LIN {X 0,Y 77.962,Z 440.495,A -85,B 0,C 180,E1 -28389.126,E2 -28389.126} C_VEL
LIN {X 0,Y 84.259,Z 435.416,A -85,B 0,C 180,E1 -28395.152,E2 -28395.152} C_VEL
LIN {X 0,Y 91.354,Z 428.999,A -85,B 0,C 180,E1 -28400.293,E2 -28400.293} C_VEL
LIN {X 0,Y 98.775,Z 421.332,A -85,B 0,C 180,E1 -28404.517,E2 -28404.517} C_VEL
LIN {X 0,Y 99.783,Z 419.685,A -85,B 0,C 180,E1 -28405.704,E2 -28405.704} C_VEL
LIN {X 0,Y 94.04,Z 422.037,A -85,B 0,C 180,E1 -28408.457,E2 -28408.457} C_VEL
LIN {X 0,Y 84.561,Z 425.489,A -85,B 0,C 180,E1 -28415.445,E2 -28415.445} C_VEL
LIN {X 0,Y 74.4,Z 429.626,A -85,B 0,C 180,E1 -28429.11,E2 -28429.11} C_VEL
LIN {X 0,Y 70.741,Z 435.431,A -85,B 0,C 180,E1 -28457.34,E2 -28457.34} C_VEL
LIN {X 0,Y 72.341,Z 436.386,A -85,B 0,C 180,E1 -28462.867,E2 -28462.867} C_VEL
LIN {X 0,Y 74.062,Z 437.713,A -85,B 0,C 180,E1 -28468.324,E2 -28468.324} C_VEL
LIN {X 0,Y 85.261,Z 440.555,A -85,B 0,C 180,E1 -28482.705,E2 -28482.705} C_VEL
LIN {X 0,Y 85.617,Z 441.316,A -85,B 0,C 180,E1 -28484.089,E2 -28484.089} C_VEL
LIN {X 0,Y 79.44,Z 445.871,A -85,B 0,C 180,E1 -28488.431,E2 -28488.431} C_VEL
LIN {X 0,Y 73.09,Z 450.242,A -85,B 0,C 180,E1 -28494.765,E2 -28494.765} C_VEL
LIN {X 0,Y 69.721,Z 452.565,A -85,B 0,C 180,E1 -28499.734,E2 -28499.734} C_VEL
LIN {X 0,Y 67.029,Z 454.469,A -85,B 0,C 180,E1 -28505.203,E2 -28505.203} C_VEL
LIN {X 0,Y 65.013,Z 455.908,A -85,B 0,C 180,E1 -28511.077,E2 -28511.077} C_VEL
LIN {X 0,Y 63.097,Z 457.574,A -85,B 0,C 180,E1 -28523.605,E2 -28523.605} C_VEL
LIN {X 0,Y 63.171,Z 457.811,A -85,B 0,C 180,E1 -28530,E2 -28530} C_VEL
LIN {X 0,Y 62.977,Z 457.55,A -85,B 0,C 180,E1 -28536.407,E2 -28536.407} C_VEL
LIN {X 0,Y 64.541,Z 455.84,A -85,B 0,C 180,E1 -28549.067,E2 -28549.067} C_VEL
LIN {X 0,Y 66.371,Z 454.364,A -85,B 0,C 180,E1 -28555.06,E2 -28555.06} C_VEL
LIN {X 0,Y 70.506,Z 451.34,A -85,B 0,C 180,E1 -28563.247,E2 -28563.247} C_VEL
LIN {X 0,Y 76.044,Z 447.27,A -85,B 0,C 180,E1 -28570.312,E2 -28570.312} C_VEL
LIN {X 0,Y 84.031,Z 441.038,A -85,B 0,C 180,E1 -28577.039,E2 -28577.039} C_VEL
LIN {X 0,Y 86.611,Z 438.899,A -85,B 0,C 180,E1 -28578.715,E2 -28578.715} C_VEL
LIN {X 0,Y 87.079,Z 437.956,A -85,B 0,C 180,E1 -28579.784,E2 -28579.784} C_VEL
LIN {X 0,Y 79.619,Z 436.48,A -85,B 0,C 180,E1 -28588.02,E2 -28588.02} C_VEL
LIN {X 0,Y 77.169,Z 435.308,A -85,B 0,C 180,E1 -28592.912,E2 -28592.912} C_VEL
LIN {X 0,Y 73.406,Z 433.371,A -85,B 0,C 180,E1 -28603.308,E2 -28603.308} C_VEL
LIN {X 0,Y 73.693,Z 429.74,A -85,B 0,C 180,E1 -28620,E2 -28620} C_VEL
LIN {X 0,Y 88.317,Z 421.829,A -85,B 0,C 180,E1 -28643.446,E2 -28643.446} C_VEL
LIN {X 0,Y 103.173,Z 415.563,A -85,B 0,C 180,E1 -28653.021,E2 -28653.021} C_VEL
LIN {X 0,Y 101.741,Z 417.578,A -85,B 0,C 180,E1 -28654.011,E2 -28654.011} C_VEL
LIN {X 0,Y 93.912,Z 426.276,A -85,B 0,C 180,E1 -28658.207,E2 -28658.207} C_VEL
LIN {X 0,Y 89.203,Z 430.846,A -85,B 0,C 180,E1 -28661.199,E2 -28661.199} C_VEL
LIN {X 0,Y 85.408,Z 433.951,A -85,B 0,C 180,E1 -28663.392,E2 -28663.392} C_VEL
LIN {X 0,Y 77.909,Z 438.596,A -85,B 0,C 180,E1 -28666.616,E2 -28666.616} C_VEL
LIN {X 0,Y 70.452,Z 442.536,A -85,B 0,C 180,E1 -28670.669,E2 -28670.669} C_VEL
LIN {X 0,Y 66.915,Z 444.545,A -85,B 0,C 180,E1 -28674.23,E2 -28674.23} C_VEL
LIN {X 0,Y 61.91,Z 447.609,A -85,B 0,C 180,E1 -28682.994,E2 -28682.994} C_VEL
LIN {X 0,Y 59.524,Z 449.005,A -85,B 0,C 180,E1 -28689.255,E2 -28689.255} C_VEL
LIN {X 0,Y 57.76,Z 449.987,A -85,B 0,C 180,E1 -28695.916,E2 -28695.916} C_VEL
LIN {X 0,Y 56.313,Z 450.815,A -85,B 0,C 180,E1 -28710,E2 -28710} C_VEL
LIN {X 0,Y 56.662,Z 450.615,A -85,B 0,C 180,E1 -28717.125,E2 -28717.125} C_VEL
LIN {X 0,Y 57.758,Z 450.026,A -85,B 0,C 180,E1 -28724.085,E2 -28724.085} C_VEL
LIN {X 0,Y 59.479,Z 449.063,A -85,B 0,C 180,E1 -28730.762,E2 -28730.762} C_VEL
LIN {X 0,Y 61.849,Z 447.699,A -85,B 0,C 180,E1 -28737.035,E2 -28737.035} C_VEL
LIN {X 0,Y 66.64,Z 444.824,A -85,B 0,C 180,E1 -28745.454,E2 -28745.454} C_VEL
LIN {X 0,Y 72.59,Z 440.908,A -85,B 0,C 180,E1 -28752.666,E2 -28752.666} C_VEL
LIN {X 0,Y 79.422,Z 435.826,A -85,B 0,C 180,E1 -28758.778,E2 -28758.778} C_VEL
LIN {X 0,Y 86.994,Z 429.408,A -85,B 0,C 180,E1 -28763.889,E2 -28763.889} C_VEL
LIN {X 0,Y 88.776,Z 427.801,A -85,B 0,C 180,E1 -28764.882,E2 -28764.882} C_VEL
LIN {X 0,Y 89.809,Z 426.453,A -85,B 0,C 180,E1 -28766.067,E2 -28766.067} C_VEL
LIN {X 0,Y 77.142,Z 430.533,A -85,B 0,C 180,E1 -28775.651,E2 -28775.651} C_VEL
LIN {X 0,Y 66.265,Z 434.834,A -85,B 0,C 180,E1 -28793.912,E2 -28793.912} C_VEL
LIN {X 0,Y 68.672,Z 441.312,A -85,B 0,C 180,E1 -28830.778,E2 -28830.778} C_VEL
LIN {X 0,Y 75.605,Z 442.948,A -85,B 0,C 180,E1 -28840.594,E2 -28840.594} C_VEL
LIN {X 0,Y 76.773,Z 443.733,A -85,B 0,C 180,E1 -28842.917,E2 -28842.917} C_VEL
LIN {X 0,Y 69.583,Z 448.493,A -85,B 0,C 180,E1 -28848.965,E2 -28848.965} C_VEL
LIN {X 0,Y 63.675,Z 452.15,A -85,B 0,C 180,E1 -28856.505,E2 -28856.505} C_VEL
LIN {X 0,Y 60.649,Z 454.053,A -85,B 0,C 180,E1 -28862.386,E2 -28862.386} C_VEL
LIN {X 0,Y 58.345,Z 455.493,A -85,B 0,C 180,E1 -28868.816,E2 -28868.816} C_VEL
LIN {X 0,Y 56.039,Z 457.158,A -85,B 0,C 180,E1 -28882.795,E2 -28882.795} C_VEL
LIN {X 0,Y 56.073,Z 457.395,A -85,B 0,C 180,E1 -28890,E2 -28890} C_VEL
LIN {X 0,Y 55.912,Z 457.133,A -85,B 0,C 180,E1 -28897.221,E2 -28897.221} C_VEL
LIN {X 0,Y 57.849,Z 455.422,A -85,B 0,C 180,E1 -28911.375,E2 -28911.375} C_VEL
LIN {X 0,Y 59.973,Z 453.945,A -85,B 0,C 180,E1 -28917.953,E2 -28917.953} C_VEL
LIN {X 0,Y 64.68,Z 450.924,A -85,B 0,C 180,E1 -28926.7,E2 -28926.7} C_VEL
LIN {X 0,Y 70.763,Z 446.853,A -85,B 0,C 180,E1 -28934.045,E2 -28934.045} C_VEL
LIN {X 0,Y 77.918,Z 441.734,A -85,B 0,C 180,E1 -28939.843,E2 -28939.843} C_VEL
LIN {X 0,Y 78.192,Z 440.975,A -85,B 0,C 180,E1 -28941.011,E2 -28941.011} C_VEL
LIN {X 0,Y 74.5,Z 440.2,A -85,B 0,C 180,E1 -28945.527,E2 -28945.527} C_VEL
LIN {X 0,Y 66.846,Z 436.213,A -85,B 0,C 180,E1 -28967.862,E2 -28967.862} C_VEL
LIN {X 0,Y 67.704,Z 433.913,A -85,B 0,C 180,E1 -28980,E2 -28980} C_VEL
LIN {X 0,Y 79.471,Z 427.848,A -85,B 0,C 180,E1 -29001.484,E2 -29001.484} C_VEL
LIN {X 0,Y 88.577,Z 424.457,A -85,B 0,C 180,E1 -29009.216,E2 -29009.216} C_VEL
LIN {X 0,Y 93.109,Z 422.662,A -85,B 0,C 180,E1 -29011.896,E2 -29011.896} C_VEL
LIN {X 0,Y 92.428,Z 424.025,A -85,B 0,C 180,E1 -29013.237,E2 -29013.237} C_VEL
LIN {X 0,Y 84.454,Z 431.482,A -85,B 0,C 180,E1 -29017.761,E2 -29017.761} C_VEL
LIN {X 0,Y 77.146,Z 437.451,A -85,B 0,C 180,E1 -29023.214,E2 -29023.214} C_VEL
LIN {X 0,Y 70.515,Z 442.168,A -85,B 0,C 180,E1 -29029.621,E2 -29029.621} C_VEL
LIN {X 0,Y 66.915,Z 444.545,A -85,B 0,C 180,E1 -29034.23,E2 -29034.23} C_VEL
LIN {X 0,Y 63.619,Z 446.327,A -85,B 0,C 180,E1 -29038.239,E2 -29038.239} C_VEL
LIN {X 0,Y 57.223,Z 448.651,A -85,B 0,C 180,E1 -29045.088,E2 -29045.088} C_VEL
LIN {X 0,Y 52.565,Z 450.064,A -85,B 0,C 180,E1 -29051.716,E2 -29051.716} C_VEL
LIN {X 0,Y 50.038,Z 450.83,A -85,B 0,C 180,E1 -29058.873,E2 -29058.873} C_VEL
LIN {X 0,Y 49.868,Z 450.864,A -85,B 0,C 180,E1 -29059.987,E2 -29059.987} C_VEL
LIN {X 0,Y 49.322,Z 451.164,A -85,B 0,C 180,E1 -29074.082,E2 -29074.082} C_VEL
LIN {X 0,Y 50.919,Z 450.441,A -85,B 0,C 180,E1 -29086.025,E2 -29086.025} C_VEL
LIN {X 0,Y 52.911,Z 449.477,A -85,B 0,C 180,E1 -29093.483,E2 -29093.483} C_VEL
LIN {X 0,Y 55.633,Z 448.112,A -85,B 0,C 180,E1 -29100.352,E2 -29100.352} C_VEL
LIN {X 0,Y 61.005,Z 445.237,A -85,B 0,C 180,E1 -29109.318,E2 -29109.318} C_VEL
LIN {X 0,Y 67.54,Z 441.321,A -85,B 0,C 180,E1 -29116.752,E2 -29116.752} C_VEL
LIN {X 0,Y 74.945,Z 436.237,A -85,B 0,C 180,E1 -29122.853,E2 -29122.853} C_VEL
LIN {X 0,Y 78.943,Z 433.189,A -85,B 0,C 180,E1 -29125.47,E2 -29125.47} C_VEL
LIN {X 0,Y 79.597,Z 432.225,A -85,B 0,C 180,E1 -29126.908,E2 -29126.908} C_VEL
LIN {X 0,Y 68.902,Z 435.279,A -85,B 0,C 180,E1 -29136.635,E2 -29136.635} C_VEL
LIN {X 0,Y 57.879,Z 441.553,A -85,B 0,C 180,E1 -29174.055,E2 -29174.055} C_VEL
LIN {X 0,Y 63.243,Z 444.517,A -85,B 0,C 180,E1 -29193.754,E2 -29193.754} C_VEL
LIN {X 0,Y 67.631,Z 445.456,A -85,B 0,C 180,E1 -29200.255,E2 -29200.255} C_VEL
LIN {X 0,Y 66.833,Z 446.644,A -85,B 0,C 180,E1 -29202.599,E2 -29202.599} C_VEL
LIN {X 0,Y 59.883,Z 450.655,A -85,B 0,C 180,E1 -29209.797,E2 -29209.797} C_VEL
LIN {X 0,Y 54.436,Z 453.637,A -85,B 0,C 180,E1 -29218.908,E2 -29218.908} C_VEL
LIN {X 0,Y 51.768,Z 455.077,A -85,B 0,C 180,E1 -29225.966,E2 -29225.966} C_VEL
LIN {X 0,Y 49.953,Z 456.106,A -85,B 0,C 180,E1 -29233.657,E2 -29233.657} C_VEL
LIN {X 0,Y 48.992,Z 456.742,A -85,B 0,C 180,E1 -29241.752,E2 -29241.752} C_VEL
LIN {X 0,Y 48.958,Z 456.979,A -85,B 0,C 180,E1 -29250,E2 -29250} C_VEL
LIN {X 0,Y 48.85,Z 456.716,A -85,B 0,C 180,E1 -29258.272,E2 -29258.272} C_VEL
LIN {X 0,Y 51.266,Z 455.004,A -85,B 0,C 180,E1 -29274.284,E2 -29274.284} C_VEL
LIN {X 0,Y 53.767,Z 453.526,A -85,B 0,C 180,E1 -29281.524,E2 -29281.524} C_VEL
LIN {X 0,Y 59.139,Z 450.508,A -85,B 0,C 180,E1 -29290.815,E2 -29290.815} C_VEL
LIN {X 0,Y 65.834,Z 446.436,A -85,B 0,C 180,E1 -29298.355,E2 -29298.355} C_VEL
LIN {X 0,Y 67.932,Z 445.077,A -85,B 0,C 180,E1 -29300.149,E2 -29300.149} C_VEL
LIN {X 0,Y 69.391,Z 443.577,A -85,B 0,C 180,E1 -29302.578,E2 -29302.578} C_VEL
LIN {X 0,Y 60.743,Z 439.877,A -85,B 0,C 180,E1 -29326.621,E2 -29326.621} C_VEL
LIN {X 0,Y 61.47,Z 437.706,A -85,B 0,C 180,E1 -29340,E2 -29340} C_VEL
LIN {X 0,Y 77.657,Z 430.826,A -85,B 0,C 180,E1 -29366.905,E2 -29366.905} C_VEL
LIN {X 0,Y 82.569,Z 429.212,A -85,B 0,C 180,E1 -29370.711,E2 -29370.711} C_VEL
LIN {X 0,Y 83.06,Z 429.58,A -85,B 0,C 180,E1 -29372.205,E2 -29372.205} C_VEL
LIN {X 0,Y 75.013,Z 436.037,A -85,B 0,C 180,E1 -29377.215,E2 -29377.215} C_VEL
LIN {X 0,Y 67.597,Z 441.161,A -85,B 0,C 180,E1 -29383.299,E2 -29383.299} C_VEL
LIN {X 0,Y 61.052,Z 445.118,A -85,B 0,C 180,E1 -29390.718,E2 -29390.718} C_VEL
LIN {X 0,Y 55.681,Z 448.025,A -85,B 0,C 180,E1 -29399.677,E2 -29399.677} C_VEL
LIN {X 0,Y 52.966,Z 449.42,A -85,B 0,C 180,E1 -29406.542,E2 -29406.542} C_VEL
LIN {X 0,Y 49.868,Z 450.864,A -85,B 0,C 180,E1 -29419.987,E2 -29419.987} C_VEL
LIN {X 0,Y 48.641,Z 451.264,A -85,B 0,C 180,E1 -29426.696,E2 -29426.696} C_VEL
LIN {X 0,Y 46.119,Z 451.387,A -85,B 0,C 180,E1 -29438.326,E2 -29438.326} C_VEL
LIN {X 0,Y 45.232,Z 450.886,A -85,B 0,C 180,E1 -29448.299,E2 -29448.299} C_VEL
LIN {X 0,Y 46.124,Z 450.089,A -85,B 0,C 180,E1 -29455.631,E2 -29455.631} C_VEL
LIN {X 0,Y 46.809,Z 449.734,A -85,B 0,C 180,E1 -29457.89,E2 -29457.89} C_VEL
LIN {X 0,Y 49.659,Z 448.525,A -85,B 0,C 180,E1 -29464.479,E2 -29464.479} C_VEL
LIN {X 0,Y 55.699,Z 445.65,A -85,B 0,C 180,E1 -29473.946,E2 -29473.946} C_VEL
LIN {X 0,Y 62.893,Z 441.733,A -85,B 0,C 180,E1 -29481.464,E2 -29481.464} C_VEL
LIN {X 0,Y 68.149,Z 438.461,A -85,B 0,C 180,E1 -29485.59,E2 -29485.59} C_VEL
LIN {X 0,Y 69.372,Z 437.247,A -85,B 0,C 180,E1 -29487.937,E2 -29487.937} C_VEL
LIN {X 0,Y 53.652,Z 441.789,A -85,B 0,C 180,E1 -29512.473,E2 -29512.473} C_VEL
LIN {X 0,Y 57.893,Z 447.352,A -85,B 0,C 180,E1 -29557.371,E2 -29557.371} C_VEL
LIN {X 0,Y 58.45,Z 448.31,A -85,B 0,C 180,E1 -29561.036,E2 -29561.036} C_VEL
LIN {X 0,Y 52.403,Z 451.32,A -85,B 0,C 180,E1 -29567.889,E2 -29567.889} C_VEL
LIN {X 0,Y 48.48,Z 453.222,A -85,B 0,C 180,E1 -29574.559,E2 -29574.559} C_VEL
LIN {X 0,Y 45.365,Z 454.661,A -85,B 0,C 180,E1 -29582.305,E2 -29582.305} C_VEL
LIN {X 0,Y 41.987,Z 456.327,A -85,B 0,C 180,E1 -29600.364,E2 -29600.364} C_VEL
LIN {X 0,Y 41.848,Z 456.562,A -85,B 0,C 180,E1 -29610,E2 -29610} C_VEL
LIN {X 0,Y 41.813,Z 456.298,A -85,B 0,C 180,E1 -29619.676,E2 -29619.676} C_VEL
LIN {X 0,Y 44.843,Z 454.585,A -85,B 0,C 180,E1 -29638.046,E2 -29638.046} C_VEL
LIN {X 0,Y 47.828,Z 453.108,A -85,B 0,C 180,E1 -29646,E2 -29646} C_VEL
LIN {X 0,Y 53.946,Z 450.09,A -85,B 0,C 180,E1 -29655.769,E2 -29655.769} C_VEL
LIN {X 0,Y 61.336,Z 446.019,A -85,B 0,C 180,E1 -29663.329,E2 -29663.329} C_VEL
LIN {X 0,Y 60.822,Z 445.728,A -85,B 0,C 180,E1 -29664.708,E2 -29664.708} C_VEL
LIN {X 0,Y 54.466,Z 443.139,A -85,B 0,C 180,E1 -29685.045,E2 -29685.045} C_VEL
LIN {X 0,Y 56.972,Z 439.97,A -85,B 0,C 180,E1 -29707.086,E2 -29707.086} C_VEL
LIN {X 0,Y 72.893,Z 434.575,A -85,B 0,C 180,E1 -29729.803,E2 -29729.803} C_VEL
LIN {X 0,Y 73.724,Z 434.479,A -85,B 0,C 180,E1 -29730.912,E2 -29730.912} C_VEL
LIN {X 0,Y 65.538,Z 439.997,A -85,B 0,C 180,E1 -29736.461,E2 -29736.461} C_VEL
LIN {X 0,Y 58.037,Z 444.321,A -85,B 0,C 180,E1 -29743.4,E2 -29743.4} C_VEL
LIN {X 0,Y 53.59,Z 446.592,A -85,B 0,C 180,E1 -29749.026,E2 -29749.026} C_VEL
LIN {X 0,Y 49.696,Z 448.44,A -85,B 0,C 180,E1 -29755.55,E2 -29755.55} C_VEL
LIN {X 0,Y 46.549,Z 449.835,A -85,B 0,C 180,E1 -29763.067,E2 -29763.067} C_VEL
LIN {X 0,Y 42.667,Z 451.419,A -85,B 0,C 180,E1 -29780.519,E2 -29780.519} C_VEL
LIN {X 0,Y 42.169,Z 451.644,A -85,B 0,C 180,E1 -29790,E2 -29790} C_VEL
LIN {X 0,Y 42.667,Z 451.443,A -85,B 0,C 180,E1 -29799.481,E2 -29799.481} C_VEL
LIN {X 0,Y 44.144,Z 450.855,A -85,B 0,C 180,E1 -29808.567,E2 -29808.567} C_VEL
LIN {X 0,Y 46.809,Z 449.734,A -85,B 0,C 180,E1 -29817.89,E2 -29817.89} C_VEL
LIN {X 0,Y 49.84,Z 448.215,A -85,B 0,C 180,E1 -29826.336,E2 -29826.336} C_VEL
LIN {X 0,Y 52.833,Z 446.326,A -85,B 0,C 180,E1 -29834.257,E2 -29834.257} C_VEL
LIN {X 0,Y 57.724,Z 442.883,A -85,B 0,C 180,E1 -29845.026,E2 -29845.026} C_VEL
LIN {X 0,Y 59.527,Z 441.545,A -85,B 0,C 180,E1 -29848.253,E2 -29848.253} C_VEL
LIN {X 0,Y 59.758,Z 441.373,A -85,B 0,C 180,E1 -29848.639,E2 -29848.639} C_VEL
LIN {X 0,Y 45.114,Z 447.337,A -85,B 0,C 180,E1 -29898.153,E2 -29898.153} C_VEL
LIN {X 0,Y 50.034,Z 449.207,A -85,B 0,C 180,E1 -29916.623,E2 -29916.623} C_VEL
LIN {X 0,Y 49.254,Z 450.098,A -85,B 0,C 180,E1 -29919.884,E2 -29919.884} C_VEL
LIN {X 0,Y 42.886,Z 452.807,A -85,B 0,C 180,E1 -29929.042,E2 -29929.042} C_VEL
LIN {X 0,Y 39.214,Z 454.246,A -85,B 0,C 180,E1 -29937.475,E2 -29937.475} C_VEL
LIN {X 0,Y 35,Z 455.911,A -85,B 0,C 180,E1 -29958.416,E2 -29958.416} C_VEL
LIN {X 0,Y 34.735,Z 456.146,A -85,B 0,C 180,E1 -29970,E2 -29970} C_VEL
LIN {X 0,Y 34.799,Z 455.88,A -85,B 0,C 180,E1 -29981.651,E2 -29981.651} C_VEL
LIN {X 0,Y 36.154,Z 455.22,A -85,B 0,C 180,E1 -29992.879,E2 -29992.879} C_VEL
LIN {X 0,Y 38.684,Z 454.166,A -85,B 0,C 180,E1 -30003.027,E2 -30003.027} C_VEL
LIN {X 0,Y 42.264,Z 452.69,A -85,B 0,C 180,E1 -30011.694,E2 -30011.694} C_VEL
LIN {X 0,Y 49.245,Z 449.673,A -85,B 0,C 180,E1 -30021.715,E2 -30021.715} C_VEL
LIN {X 0,Y 51.867,Z 448.425,A -85,B 0,C 180,E1 -30024.39,E2 -30024.39} C_VEL
LIN {X 0,Y 52.156,Z 447.663,A -85,B 0,C 180,E1 -30027.385,E2 -30027.385} C_VEL
LIN {X 0,Y 47.72,Z 445.115,A -85,B 0,C 180,E1 -30051.531,E2 -30051.531} C_VEL
LIN {X 0,Y 50.409,Z 443.136,A -85,B 0,C 180,E1 -30068.015,E2 -30068.015} C_VEL
LIN {X 0,Y 62.85,Z 439.298,A -85,B 0,C 180,E1 -30088.53,E2 -30088.53} C_VEL
LIN {X 0,Y 61.006,Z 440.737,A -85,B 0,C 180,E1 -30091.553,E2 -30091.553} C_VEL
LIN {X 0,Y 50.873,Z 445.948,A -85,B 0,C 180,E1 -30100.553,E2 -30100.553} C_VEL
LIN {X 0,Y 44.045,Z 448.854,A -85,B 0,C 180,E1 -30110.338,E2 -30110.338} C_VEL
LIN {X 0,Y 40.348,Z 450.251,A -85,B 0,C 180,E1 -30118.496,E2 -30118.496} C_VEL
LIN {X 0,Y 37.517,Z 451.231,A -85,B 0,C 180,E1 -30127.997,E2 -30127.997} C_VEL
LIN {X 0,Y 35.103,Z 452.057,A -85,B 0,C 180,E1 -30150,E2 -30150} C_VEL
LIN {X 0,Y 35.695,Z 451.857,A -85,B 0,C 180,E1 -30161.355,E2 -30161.355} C_VEL
LIN {X 0,Y 37.497,Z 451.27,A -85,B 0,C 180,E1 -30172.015,E2 -30172.015} C_VEL
LIN {X 0,Y 40.491,Z 450.228,A -85,B 0,C 180,E1 -30182.049,E2 -30182.049} C_VEL
LIN {X 0,Y 43.998,Z 448.939,A -85,B 0,C 180,E1 -30189.713,E2 -30189.713} C_VEL
LIN {X 0,Y 50.836,Z 446.063,A -85,B 0,C 180,E1 -30199.497,E2 -30199.497} C_VEL
LIN {X 0,Y 58.74,Z 442.146,A -85,B 0,C 180,E1 -30206.879,E2 -30206.879} C_VEL
LIN {X 0,Y 59.527,Z 441.545,A -85,B 0,C 180,E1 -30208.253,E2 -30208.253} C_VEL
LIN {X 0,Y 59.753,Z 441.142,A -85,B 0,C 180,E1 -30209.908,E2 -30209.908} C_VEL
LIN {X 0,Y 58.581,Z 441.184,A -85,B 0,C 180,E1 -30212.673,E2 -30212.673} C_VEL
LIN {X 0,Y 55.263,Z 442.123,A -85,B 0,C 180,E1 -30216.276,E2 -30216.276} C_VEL
LIN {X 0,Y 52.346,Z 443.094,A -85,B 0,C 180,E1 -30218.634,E2 -30218.634} C_VEL
LIN {X 0,Y 42.673,Z 446.419,A -85,B 0,C 180,E1 -30227.38,E2 -30227.38} C_VEL
LIN {X 0,Y 39.914,Z 447.373,A -85,B 0,C 180,E1 -30232.832,E2 -30232.832} C_VEL
LIN {X 0,Y 39.084,Z 447.715,A -85,B 0,C 180,E1 -30236.124,E2 -30236.124} C_VEL
LIN {X 0,Y 41.437,Z 450.606,A -85,B 0,C 180,E1 -30273.779,E2 -30273.779} C_VEL
LIN {X 0,Y 40.178,Z 451.533,A -85,B 0,C 180,E1 -30278.468,E2 -30278.468} C_VEL
LIN {X 0,Y 33.426,Z 453.83,A -85,B 0,C 180,E1 -30290.892,E2 -30290.892} C_VEL
LIN {X 0,Y 28.092,Z 455.496,A -85,B 0,C 180,E1 -30315.512,E2 -30315.512} C_VEL
LIN {X 0,Y 27.633,Z 455.73,A -85,B 0,C 180,E1 -30330,E2 -30330} C_VEL
LIN {X 0,Y 27.867,Z 455.464,A -85,B 0,C 180,E1 -30344.608,E2 -30344.608} C_VEL
LIN {X 0,Y 32.934,Z 453.748,A -85,B 0,C 180,E1 -30369.807,E2 -30369.807} C_VEL
LIN {X 0,Y 37.242,Z 452.272,A -85,B 0,C 180,E1 -30379.012,E2 -30379.012} C_VEL
LIN {X 0,Y 43.574,Z 449.892,A -85,B 0,C 180,E1 -30387.242,E2 -30387.242} C_VEL
LIN {X 0,Y 43.586,Z 449.29,A -85,B 0,C 180,E1 -30391.071,E2 -30391.071} C_VEL
LIN {X 0,Y 42.236,Z 446.516,A -85,B 0,C 180,E1 -30423.241,E2 -30423.241} C_VEL
LIN {X 0,Y 52.454,Z 443.435,A -85,B 0,C 180,E1 -30446.478,E2 -30446.478} C_VEL
LIN {X 0,Y 52.649,Z 443.643,A -85,B 0,C 180,E1 -30448.777,E2 -30448.777} C_VEL
LIN {X 0,Y 43.877,Z 447.423,A -85,B 0,C 180,E1 -30456.786,E2 -30456.786} C_VEL
LIN {X 0,Y 38.852,Z 449.27,A -85,B 0,C 180,E1 -30463.65,E2 -30463.65} C_VEL
LIN {X 0,Y 34.511,Z 450.666,A -85,B 0,C 180,E1 -30472.342,E2 -30472.342} C_VEL
LIN {X 0,Y 31.06,Z 451.646,A -85,B 0,C 180,E1 -30483.093,E2 -30483.093} C_VEL
LIN {X 0,Y 28.029,Z 452.471,A -85,B 0,C 180,E1 -30510,E2 -30510} C_VEL
LIN {X 0,Y 28.786,Z 452.272,A -85,B 0,C 180,E1 -30524.131,E2 -30524.131} C_VEL
LIN {X 0,Y 31.047,Z 451.684,A -85,B 0,C 180,E1 -30536.919,E2 -30536.919} C_VEL
LIN {X 0,Y 34.455,Z 450.721,A -85,B 0,C 180,E1 -30547.73,E2 -30547.73} C_VEL
LIN {X 0,Y 38.802,Z 449.354,A -85,B 0,C 180,E1 -30556.427,E2 -30556.427} C_VEL
LIN {X 0,Y 46.549,Z 446.476,A -85,B 0,C 180,E1 -30566.14,E2 -30566.14} C_VEL
LIN {X 0,Y 49.345,Z 445.27,A -85,B 0,C 180,E1 -30568.712,E2 -30568.712} C_VEL
LIN {X 0,Y 46.695,Z 445.595,A -85,B 0,C 180,E1 -30574.564,E2 -30574.564} C_VEL
LIN {X 0,Y 39.084,Z 447.715,A -85,B 0,C 180,E1 -30596.124,E2 -30596.124} C_VEL
LIN {X 0,Y 37.703,Z 448.357,A -85,B 0,C 180,E1 -30601.611,E2 -30601.611} C_VEL
LIN {X 0,Y 32.406,Z 451.103,A -85,B 0,C 180,E1 -30621.527,E2 -30621.527} C_VEL
LIN {X 0,Y 32.651,Z 451.677,A -85,B 0,C 180,E1 -30628.479,E2 -30628.479} C_VEL
LIN {X 0,Y 33.475,Z 451.977,A -85,B 0,C 180,E1 -30632.88,E2 -30632.88} C_VEL
LIN {X 0,Y 28.263,Z 453.414,A -85,B 0,C 180,E1 -30641.756,E2 -30641.756} C_VEL
LIN {X 0,Y 21.277,Z 455.08,A -85,B 0,C 180,E1 -30670.713,E2 -30670.713} C_VEL
LIN {X 0,Y 20.522,Z 455.314,A -85,B 0,C 180,E1 -30690,E2 -30690} C_VEL
LIN {X 0,Y 21.049,Z 455.046,A -85,B 0,C 180,E1 -30709.505,E2 -30709.505} C_VEL
LIN {X 0,Y 27.837,Z 453.331,A -85,B 0,C 180,E1 -30739.237,E2 -30739.237} C_VEL
LIN {X 0,Y 34.726,Z 451.308,A -85,B 0,C 180,E1 -30750.528,E2 -30750.528} C_VEL
LIN {X 0,Y 35.274,Z 450.596,A -85,B 0,C 180,E1 -30756.517,E2 -30756.517} C_VEL
LIN {X 0,Y 36.922,Z 448.218,A -85,B 0,C 180,E1 -30790.974,E2 -30790.974} C_VEL
LIN {X 0,Y 42.659,Z 446.807,A -85,B 0,C 180,E1 -30804.713,E2 -30804.713} C_VEL
LIN {X 0,Y 41.445,Z 447.345,A -85,B 0,C 180,E1 -30807.355,E2 -30807.355} C_VEL
LIN {X 0,Y 34.338,Z 449.686,A -85,B 0,C 180,E1 -30815.045,E2 -30815.045} C_VEL
LIN {X 0,Y 29.214,Z 451.082,A -85,B 0,C 180,E1 -30823.805,E2 -30823.805} C_VEL
LIN {X 0,Y 24.949,Z 452.061,A -85,B 0,C 180,E1 -30835.709,E2 -30835.709} C_VEL
LIN {X 0,Y 20.941,Z 452.886,A -85,B 0,C 180,E1 -30870,E2 -30870} C_VEL
LIN {X 0,Y 21.988,Z 452.686,A -85,B 0,C 180,E1 -30888.64,E2 -30888.64} C_VEL
LIN {X 0,Y 24.939,Z 452.098,A -85,B 0,C 180,E1 -30904.306,E2 -30904.306} C_VEL
LIN {X 0,Y 29.176,Z 451.135,A -85,B 0,C 180,E1 -30916.273,E2 -30916.273} C_VEL
LIN {X 0,Y 38.13,Z 448.587,A -85,B 0,C 180,E1 -30929.593,E2 -30929.593} C_VEL
LIN {X 0,Y 39.269,Z 448.077,A -85,B 0,C 180,E1 -30932.678,E2 -30932.678} C_VEL
LIN {X 0,Y 32.651,Z 451.677,A -85,B 0,C 180,E1 -30988.479,E2 -30988.479} C_VEL
LIN {X 0,Y 32.356,Z 452.023,A -85,B 0,C 180,E1 -30991.488,E2 -30991.488} C_VEL
LIN {X 0,Y 30.74,Z 452.539,A -85,B 0,C 180,E1 -30994.733,E2 -30994.733} C_VEL
LIN {X 0,Y 27.417,Z 453.241,A -85,B 0,C 180,E1 -30998.326,E2 -30998.326} C_VEL
LIN {X 0,Y 18.472,Z 454.262,A -85,B 0,C 180,E1 -31007.013,E2 -31007.013} C_VEL
LIN {X 0,Y 15.475,Z 454.552,A -85,B 0,C 180,E1 -31016.302,E2 -31016.302} C_VEL
LIN {X 0,Y 15.07,Z 454.596,A -85,B 0,C 180,E1 -31018.936,E2 -31018.936} C_VEL
LIN {X 0,Y 13.411,Z 454.898,A -85,B 0,C 180,E1 -31050,E2 -31050} C_VEL
LIN {X 0,Y 14.524,Z 454.629,A -85,B 0,C 180,E1 -31078.94,E2 -31078.94} C_VEL
LIN {X 0,Y 23.798,Z 452.913,A -85,B 0,C 180,E1 -31112.368,E2 -31112.368} C_VEL
LIN {X 0,Y 26.111,Z 452.377,A -85,B 0,C 180,E1 -31115.812,E2 -31115.812} C_VEL
LIN {X 0,Y 27.689,Z 451.775,A -85,B 0,C 180,E1 -31121.331,E2 -31121.331} C_VEL
LIN {X 0,Y 32.196,Z 449.663,A -85,B 0,C 180,E1 -31160.413,E2 -31160.413} C_VEL
LIN {X 0,Y 30.819,Z 450.101,A -85,B 0,C 180,E1 -31164.192,E2 -31164.192} C_VEL
LIN {X 0,Y 24.843,Z 451.496,A -85,B 0,C 180,E1 -31171.93,E2 -31171.93} C_VEL
LIN {X 0,Y 19.501,Z 452.477,A -85,B 0,C 180,E1 -31183.881,E2 -31183.881} C_VEL
LIN {X 0,Y 13.861,Z 453.301,A -85,B 0,C 180,E1 -31230,E2 -31230} C_VEL
LIN {X 0,Y 15.438,Z 453.101,A -85,B 0,C 180,E1 -31257.081,E2 -31257.081} C_VEL
LIN {X 0,Y 19.492,Z 452.513,A -85,B 0,C 180,E1 -31276.146,E2 -31276.146} C_VEL
LIN {X 0,Y 27.015,Z 451.075,A -85,B 0,C 180,E1 -31291.483,E2 -31291.483} C_VEL
LIN {X 0,Y 28.998,Z 450.565,A -85,B 0,C 180,E1 -31296.69,E2 -31296.69} C_VEL
LIN {X 0,Y 24.296,Z 452.337,A -85,B 0,C 180,E1 -31336.813,E2 -31336.813} C_VEL
LIN {X 0,Y 24.121,Z 452.998,A -85,B 0,C 180,E1 -31349.06,E2 -31349.06} C_VEL
LIN {X 0,Y 15.07,Z 454.596,A -85,B 0,C 180,E1 -31378.936,E2 -31378.936} C_VEL
LIN {X 0,Y 13.024,Z 454.805,A -85,B 0,C 180,E1 -31392.598,E2 -31392.598} C_VEL
LIN {X 0,Y 10.23,Z 454.726,A -85,B 0,C 180,E1 -31415.335,E2 -31415.335} C_VEL
LIN {X 0,Y 10.135,Z 454.179,A -85,B 0,C 180,E1 -31462.828,E2 -31462.828} C_VEL
LIN {X 0,Y 12.973,Z 453.745,A -85,B 0,C 180,E1 -31477.272,E2 -31477.272} C_VEL
LIN {X 0,Y 19.333,Z 452.86,A -85,B 0,C 180,E1 -31487.558,E2 -31487.558} C_VEL
LIN {X 0,Y 20.479,Z 452.508,A -85,B 0,C 180,E1 -31493.9,E2 -31493.9} C_VEL
LIN {X 0,Y 21.165,Z 452.158,A -85,B 0,C 180,E1 -31505.024,E2 -31505.024} C_VEL
LIN {X 0,Y 21.935,Z 451.912,A -85,B 0,C 180,E1 -31516.008,E2 -31516.008} C_VEL
LIN {X 0,Y 15.462,Z 452.891,A -85,B 0,C 180,E1 -31524.619,E2 -31524.619} C_VEL
LIN {X 0,Y 9.696,Z 453.493,A -85,B 0,C 180,E1 -31543.547,E2 -31543.547} C_VEL
LIN {X 0,Y 6.781,Z 453.715,A -85,B 0,C 180,E1 -31590,E2 -31590} C_VEL
LIN {X 0,Y 9.696,Z 453.514,A -85,B 0,C 180,E1 -31636.456,E2 -31636.456} C_VEL
LIN {X 0,Y 17.223,Z 452.711,A -85,B 0,C 180,E1 -31658.575,E2 -31658.575} C_VEL
LIN {X 0,Y 18.918,Z 452.476,A -85,B 0,C 180,E1 -31665.448,E2 -31665.448} C_VEL
LIN {X 0,Y 17.162,Z 453.119,A -85,B 0,C 180,E1 -31688.833,E2 -31688.833} C_VEL
LIN {X 0,Y 16.331,Z 453.438,A -85,B 0,C 180,E1 -31698.275,E2 -31698.275} C_VEL
LIN {X 0,Y 9.16,Z 454.249,A -85,B 0,C 180,E1 -31719.896,E2 -31719.896} C_VEL
LIN {X 0,Y 6.294,Z 454.481,A -85,B 0,C 180,E1 -31770,E2 -31770} C_VEL
LIN {X 0,Y 12.973,Z 453.745,A -85,B 0,C 180,E1 -31837.272,E2 -31837.272} C_VEL
LIN {X 0,Y 14.916,Z 455.737,A -85,B 0,C 180,E1 -31841.408,E2 -31841.408} C_VEL
LIN {X 0,Y 14.916,Z 600,A -85,B 0,C 180,E1 -31841.408,E2 -31841.408} C_VEL
LIN {X 0,Y 14.916,Z 600,A -85,B 0,C 180,E1 -31841.408,E2 -31841.408}

QRS_NEXT_CUT()

QRS_NEXT()
QRS_HOME()

END
